(* Logix 5000 project; controller DEMOGUI 5069-L306ERM rev 30.11; software revision 30.00 *)

TASK MainTask (continuous, watchdog 500 ms) : MainProgram

MODULES
   Local : 5069-L306ERM (5069 0, rev 30.11)
      DIGIN : 5069-IB16 (5069 1, rev 2.1, StandardDataDriven RPI 150 ms)
      DIGOUT : 5069-OB16 (5069 3, rev 2.1, StandardDataDriven RPI 150 ms)
      ANALOGIN : vendor 1 type 115 code 314 (5069 2, rev 2.1, StandardDataDriven RPI 100 ms)
      ANALOGOUT : vendor 1 type 115 code 320 (5069 4, rev 2.1, StandardDataDriven RPI 103 ms)
END_MODULES

VAR_GLOBAL   (* controller tags *)
   DEGREES : REAL;
   THERM : ALIAS FOR Local:2:I.Ch01.Data;   // Thermister
END_VAR

PROGRAM MainProgram   (* main routine MainRoutine *)
VAR
   GL : ALIAS FOR Local:3:O.Pt01Data;   // GREEN LIGHT
   LB : BOOL;   // BREAK LATCH
   M1 : BOOL;   // ENABLE MOTOR
   MOFF : BOOL;   // Turns Motor Off
   MOTOR : ALIAS FOR Local:4:O.Ch01.Data;
   ONS1 : BOOL;
   ONY : DINT;   // TURN ON YELLOW LIGHT
   OPT : BOOL;   // OPTION: TIMER OR VIN
   PB1 : ALIAS FOR Local:1:I.Pt00Data;   // START Green LIGHT AND TIMER
   PB2 : ALIAS FOR Local:1:I.Pt01Data;   // START 20 SEC TIMER
   PT : BOOL;   // ENABLE POTENTIOMETER INPUT
   RL : ALIAS FOR Local:3:O.Pt00Data;   // RED LIGHT
   SP : REAL;   // MOTOR SPEED
   T1 : TIMER := (PRE := 30000);   // GREEN LIGHT TIMER
   T2 : TIMER := (PRE := 20000);
   TH : REAL;   // THRESHOLD
   TOGGLE : ALIAS FOR Local:1:I.Pt03Data;   // ENABLE COMPARE
   VALUE : REAL;
   VIN : ALIAS FOR Local:2:I.Ch00.Data;   // POTENTIOMETER VOLTAGE
END_VAR

ROUTINE MainRoutine   (* ladder *)
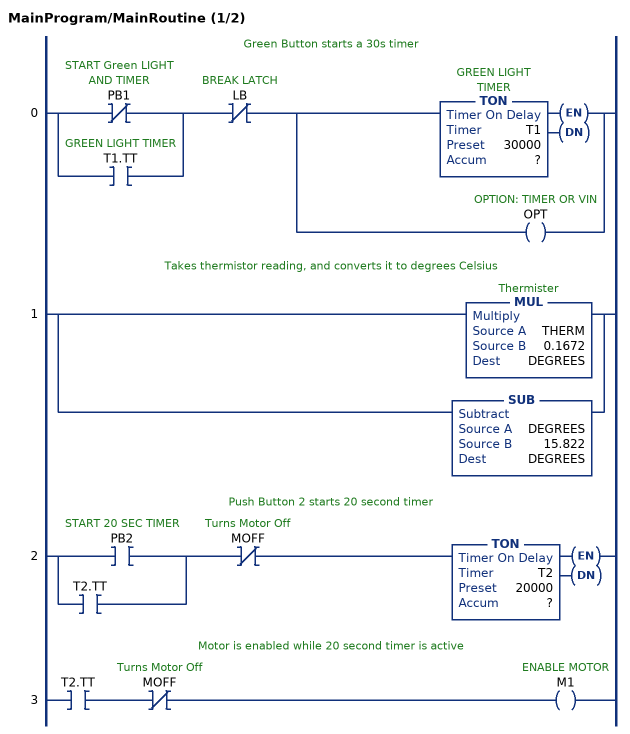
   // Green Button starts a 30s timer
   0: [XIO(PB1) ,XIC(T1.TT) ]XIO(LB)[TON(T1,?,?) ,OTE(OPT) ];
   // Takes thermistor reading, and converts it to degrees Celsius
   1: [MUL(THERM,0.1672,DEGREES) ,SUB(DEGREES,15.822,DEGREES) ];
   // Push Button 2 starts 20 second timer
   2: [XIC(PB2) ,XIC(T2.TT) ]XIO(MOFF)TON(T2,?,?);
   // Motor is enabled while 20 second timer is active
   3: XIC(T2.TT)XIO(MOFF)OTE(M1);
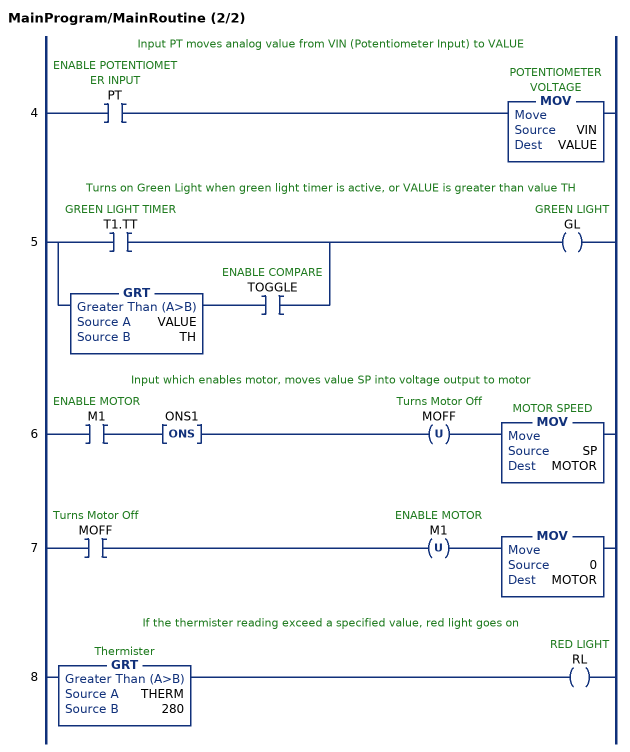
   // Input PT moves analog value from VIN (Potentiometer Input) to VALUE
   4: XIC(PT)MOV(VIN,VALUE);
   // Turns on Green Light when green light timer is active, or VALUE is greater than value TH
   5: [XIC(T1.TT) ,GRT(VALUE,TH) XIC(TOGGLE) ]OTE(GL);
   // Input which enables motor, moves value SP into voltage output to motor
   6: XIC(M1)ONS(ONS1)OTU(MOFF)MOV(SP,MOTOR);
   7: XIC(MOFF)OTU(M1)MOV(0,MOTOR);
   // If the thermister reading exceed a specified value, red light goes on
   8: GRT(THERM,280)OTE(RL);
END_ROUTINE
END_PROGRAM
